# EPICS substitutions: apps/caenHvApp/Db/seq/mvtOnOff-bmt.substitutions
file "db/mvtOnOff-bmt-1sec-1type.db"
{
pattern { SEC TYPE  PW    PWVAL}
        { 1   DRIFT pwoff 0 }
        { 2   DRIFT pwoff 0 }
        { 3   DRIFT pwoff 0 }
        { 1   STRIP pwoff 0 }
        { 2   STRIP pwoff 0 }
        { 3   STRIP pwoff 0 }
        { 1   DRIFT pwon  1 }
        { 2   DRIFT pwon  1 }
        { 3   DRIFT pwon  1 }
        { 1   STRIP pwon  1 }
        { 2   STRIP pwon  1 }
        { 3   STRIP pwon  1 }
}
